// Command that detect the execution AND generates one cycle TRUE on the output Q
FUNCTION_BLOCK PUBLIC TriggerCommand EXTENDS CommandBase
VAR_INPUT
END_VAR
VAR_OUTPUT
	Q : BOOL;
END_VAR
VAR
	bInit 	: BOOL;
END_VAR

// Will be executed in the same cycle ``stHandshake.bExecute`` changes to ``true``
METHOD PROTECTED Init
bInit := TRUE;
END_METHOD

// Execute the funktional part of the command implementation. Will be executed in the same cycle ``stHandshake.bExecute`` changes to ``true`` after the ``Init`` Method
METHOD PROTECTED Task : BOOL
// Task Code:
// dedect task completed
IF (NOT bInit AND Q) THEN
	// Task comlete;
	Task := SUPER^.Task();;
END_IF

// set output trigger
Q := bInit;

// Reset after 1. cycle
bInit := FALSE;
END_METHOD

END_FUNCTION_BLOCK

(* stored: Version 1.1.0.1, ProductVersion 3.1.4022.10
   POU TriggerCommand: Id {d02418d5-5cd7-0a17-16e2-bc96f2eeb812}, SpecialFunc None
   Method Init: Id {fefad13b-36f4-09af-2cda-4ebdb7042fe2}
   Method Task: Id {46d14659-9a33-0b69-1323-6405b400ef2f} *)
